Staubli VAL3: onStart.pgx

program onStart()
  local num i
begin
  cls()
  userPage()
  call use:nullKey(nKey)
  call buildList()
  call refreshStatic()
end
